(* PLC project Unnamed, Unknown Unnamed 1 *)
(* stored: creationDateTime 2025-11-24T11:16:17, modificationDateTime 2025-11-28T12:57:50 *)

PROGRAM Lab2
  VAR
    Potentiometer AT %IW1 : UINT := 1;
    Ljussensor AT %IW2 : UINT := 1;
  END_VAR
  VAR
    S0 : BOOL := False;
    S1 : BOOL := False;
    Light_sample : BOOL := False;
    Poten_sample : BOOL;
    Light_damaged : BOOL := False;
    Poten_damaged : BOOL := False;
    Dark : BOOL := False;
    Bright : BOOL := False;
    High : BOOL := False;
    Medium : BOOL := False;
    Low : BOOL := False;
    Damaged_comp : UINT := 0;
    Light_comp : UINT := 32768;
    High_comp : UINT := 43690;
    Low_comp : UINT := 21845;
  END_VAR
  VAR
    Relay AT %QX0.0 : BOOL := 0;
  END_VAR
  VAR
    CTU0 : CTU;
    TON0 : TON;
    T50ms : TIME := T#50ms;
    Tick_100ms : BOOL := 0;
    Fifty_ticks : INT := 50;
    TON1 : TON;
    R_TRIG0 : R_TRIG;
    F_TRIG0 : F_TRIG;
  END_VAR
  VAR  (* added by the conversion: wires and edge detectors of the diagram *)
    R_TRIG1 : R_TRIG;
    _GT34_OUT : BOOL;
    _LT35_OUT : BOOL;
    _EQ80_OUT : BOOL;
  END_VAR

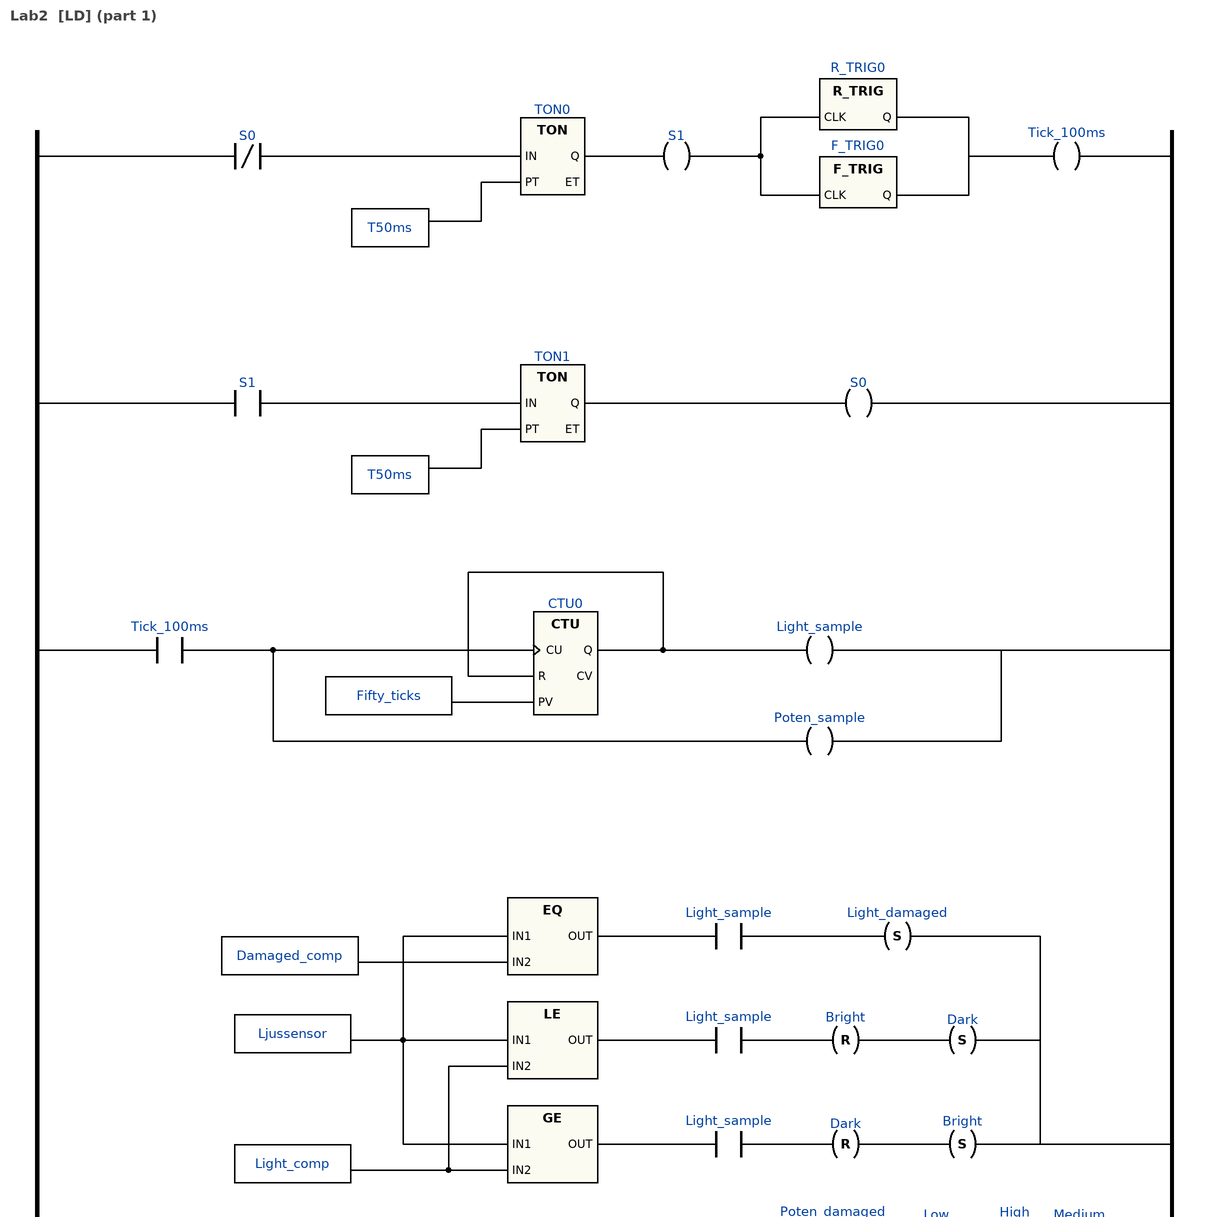
(* LD diagram, written out as Structured Text *)
TON0(IN := NOT S0, PT := T50ms);
R_TRIG0(CLK := TON0.Q);
F_TRIG0(CLK := TON0.Q);
Tick_100ms := R_TRIG0.Q OR F_TRIG0.Q;
R_TRIG1(CLK := Tick_100ms);
CTU0(CU := R_TRIG1.Q, R := CTU0.Q, PV := Fifty_ticks);
Light_sample := CTU0.Q;
TON1(IN := S1, PT := T50ms);
S0 := TON1.Q;
S1 := TON0.Q;
Poten_sample := Tick_100ms;
IF Ljussensor = Damaged_comp AND Light_sample THEN Light_damaged := TRUE; END_IF;
IF Ljussensor >= Light_comp AND Light_sample THEN Bright := TRUE; END_IF;
IF Ljussensor <= Light_comp AND Light_sample THEN Dark := TRUE; END_IF;
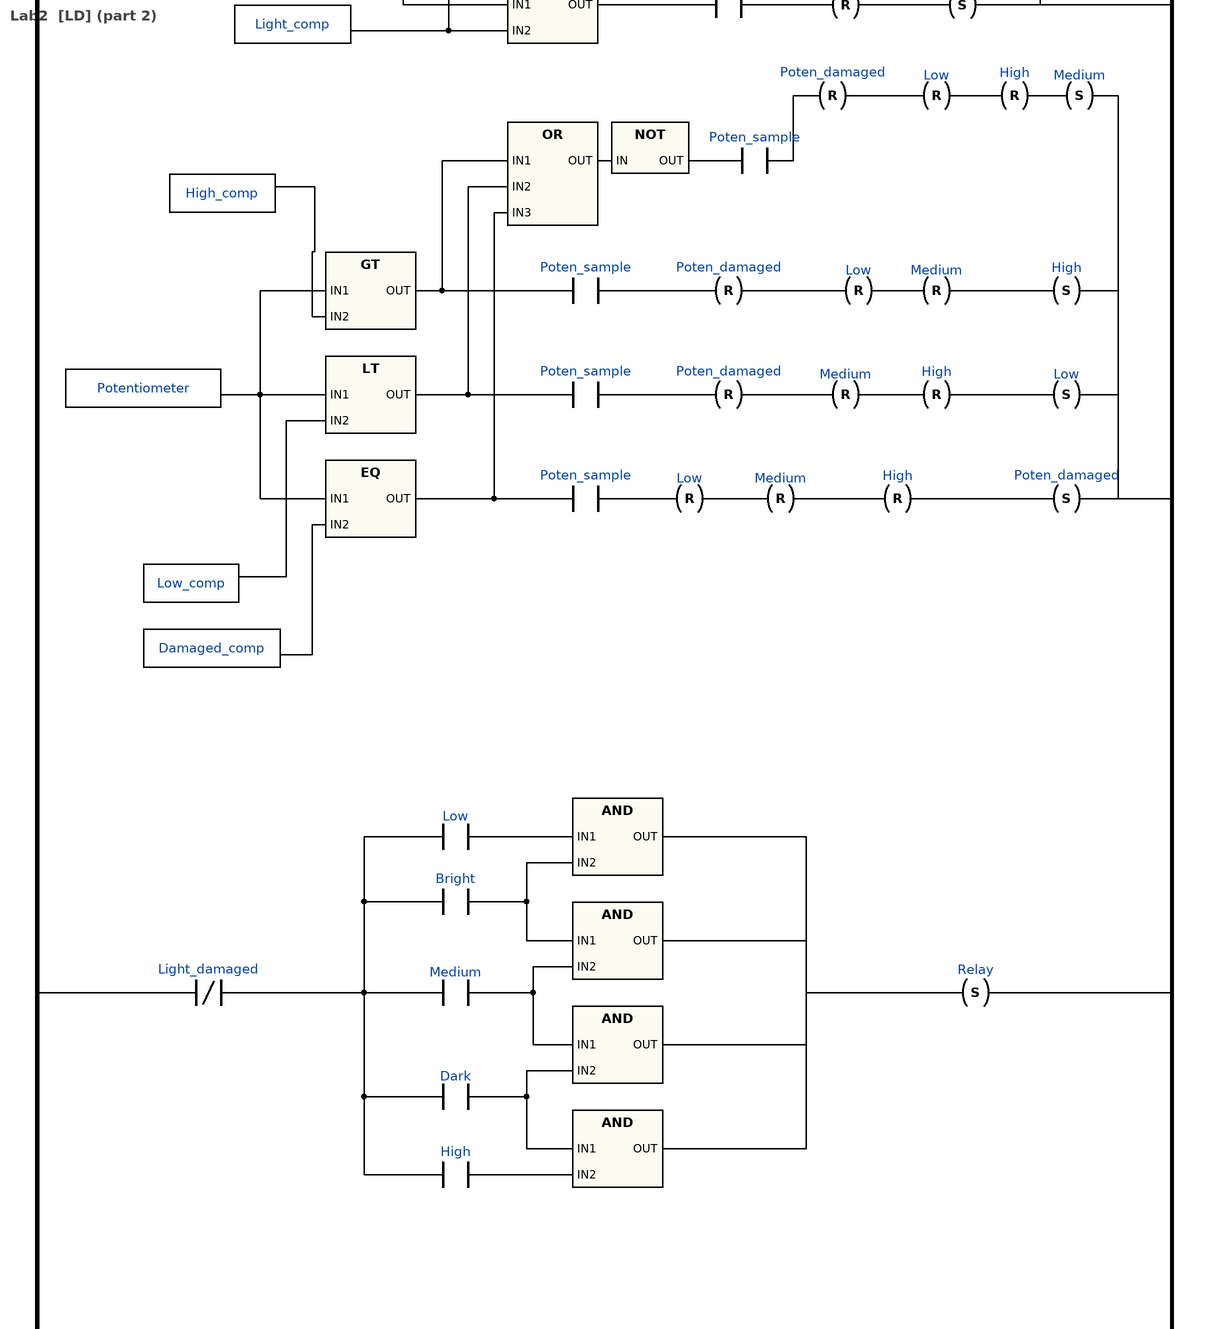
_GT34_OUT := Potentiometer > High_comp;
IF _GT34_OUT AND Poten_sample THEN High := TRUE; END_IF;
_LT35_OUT := Potentiometer < Low_comp;
IF _LT35_OUT AND Poten_sample THEN Low := TRUE; END_IF;
_EQ80_OUT := Potentiometer = Damaged_comp;
IF NOT (_GT34_OUT OR _LT35_OUT OR _EQ80_OUT) AND Poten_sample THEN Medium := TRUE; END_IF;
IF _EQ80_OUT AND Poten_sample THEN Poten_damaged := TRUE; END_IF;
IF NOT Light_damaged AND Low AND NOT Light_damaged AND Bright OR NOT Light_damaged AND Bright AND NOT Light_damaged AND Medium OR NOT Light_damaged AND Dark AND NOT Light_damaged AND High OR NOT Light_damaged AND Medium AND NOT Light_damaged AND Dark THEN Relay := TRUE; END_IF;
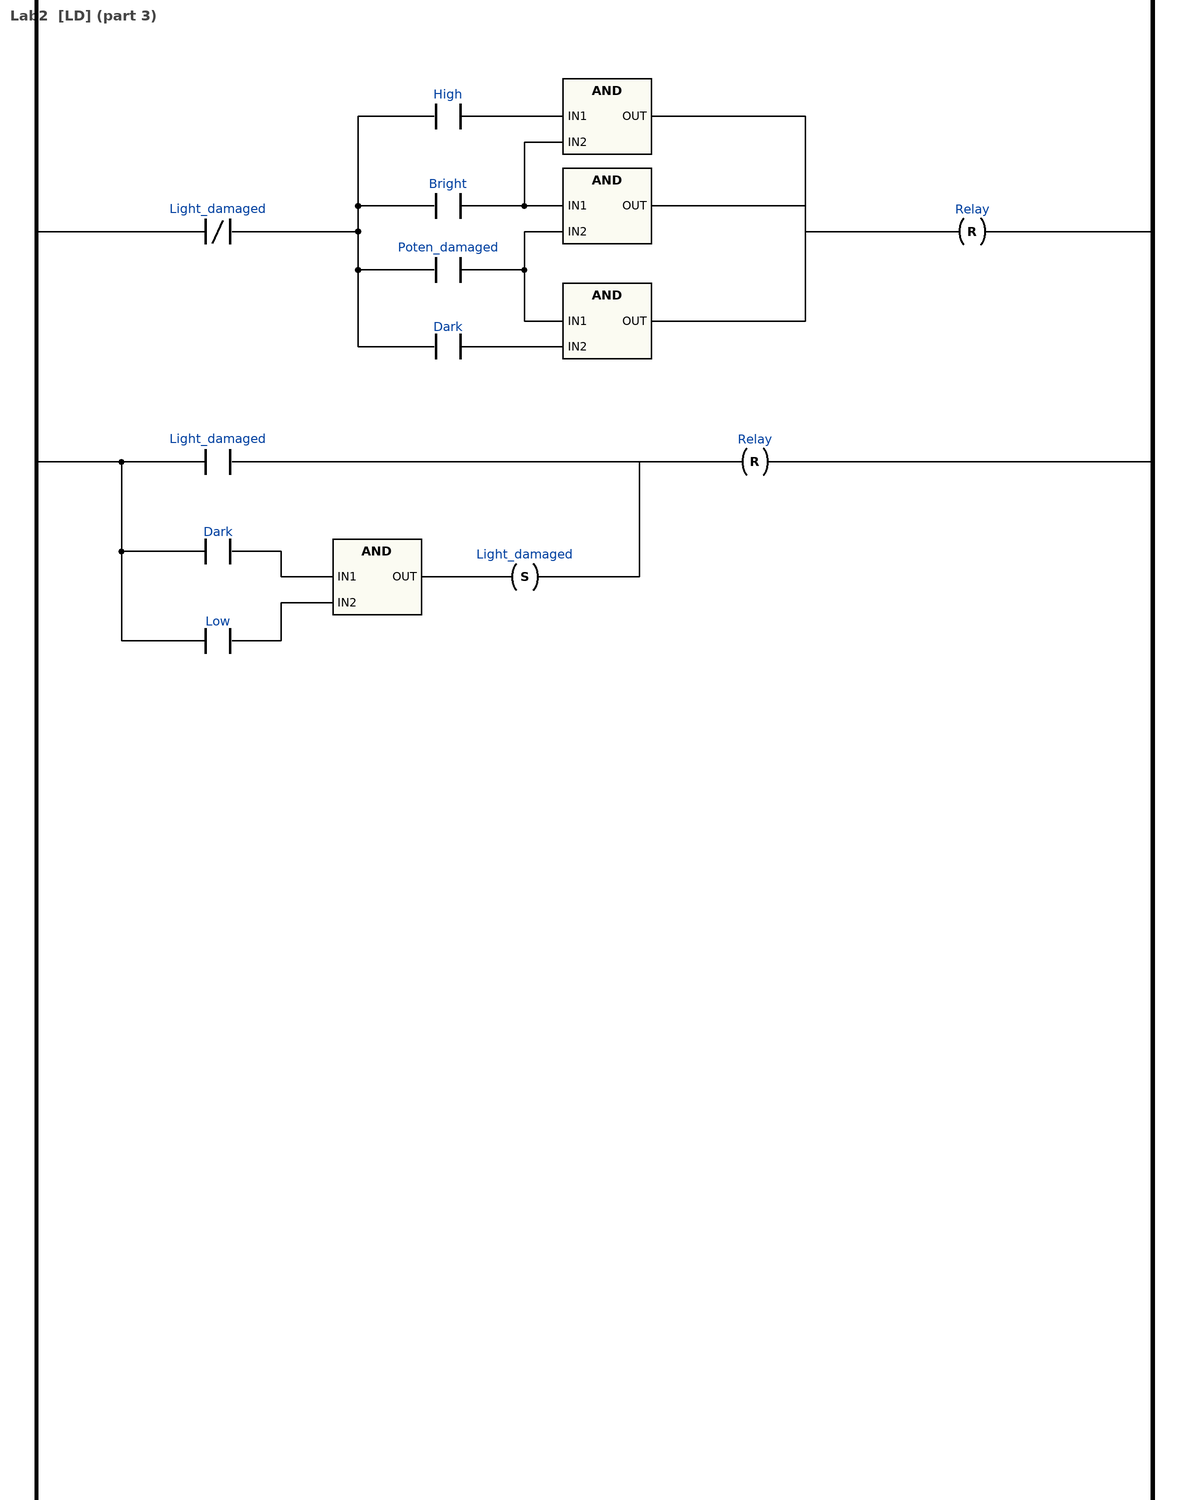
IF NOT Light_damaged AND Bright AND NOT Light_damaged AND Poten_damaged OR NOT Light_damaged AND High AND NOT Light_damaged AND Bright OR NOT Light_damaged AND Poten_damaged AND NOT Light_damaged AND Dark THEN Relay := FALSE; END_IF;
IF Light_damaged OR Dark AND Low THEN Relay := FALSE; END_IF;
IF Dark AND Low THEN Light_damaged := TRUE; END_IF;
IF Ljussensor >= Light_comp AND Light_sample THEN Dark := FALSE; END_IF;
IF Ljussensor <= Light_comp AND Light_sample THEN Bright := FALSE; END_IF;
IF _GT34_OUT AND Poten_sample THEN Poten_damaged := FALSE; END_IF;
IF _LT35_OUT AND Poten_sample THEN Poten_damaged := FALSE; END_IF;
IF NOT (_GT34_OUT OR _LT35_OUT OR _EQ80_OUT) AND Poten_sample THEN Poten_damaged := FALSE; END_IF;
IF _EQ80_OUT AND Poten_sample THEN Low := FALSE; END_IF;
IF _GT34_OUT AND Poten_sample THEN Low := FALSE; END_IF;
IF NOT (_GT34_OUT OR _LT35_OUT OR _EQ80_OUT) AND Poten_sample THEN Low := FALSE; END_IF;
IF _GT34_OUT AND Poten_sample THEN Medium := FALSE; END_IF;
IF _LT35_OUT AND Poten_sample THEN Medium := FALSE; END_IF;
IF _EQ80_OUT AND Poten_sample THEN Medium := FALSE; END_IF;
IF NOT (_GT34_OUT OR _LT35_OUT OR _EQ80_OUT) AND Poten_sample THEN High := FALSE; END_IF;
IF _LT35_OUT AND Poten_sample THEN High := FALSE; END_IF;
IF _EQ80_OUT AND Poten_sample THEN High := FALSE; END_IF;
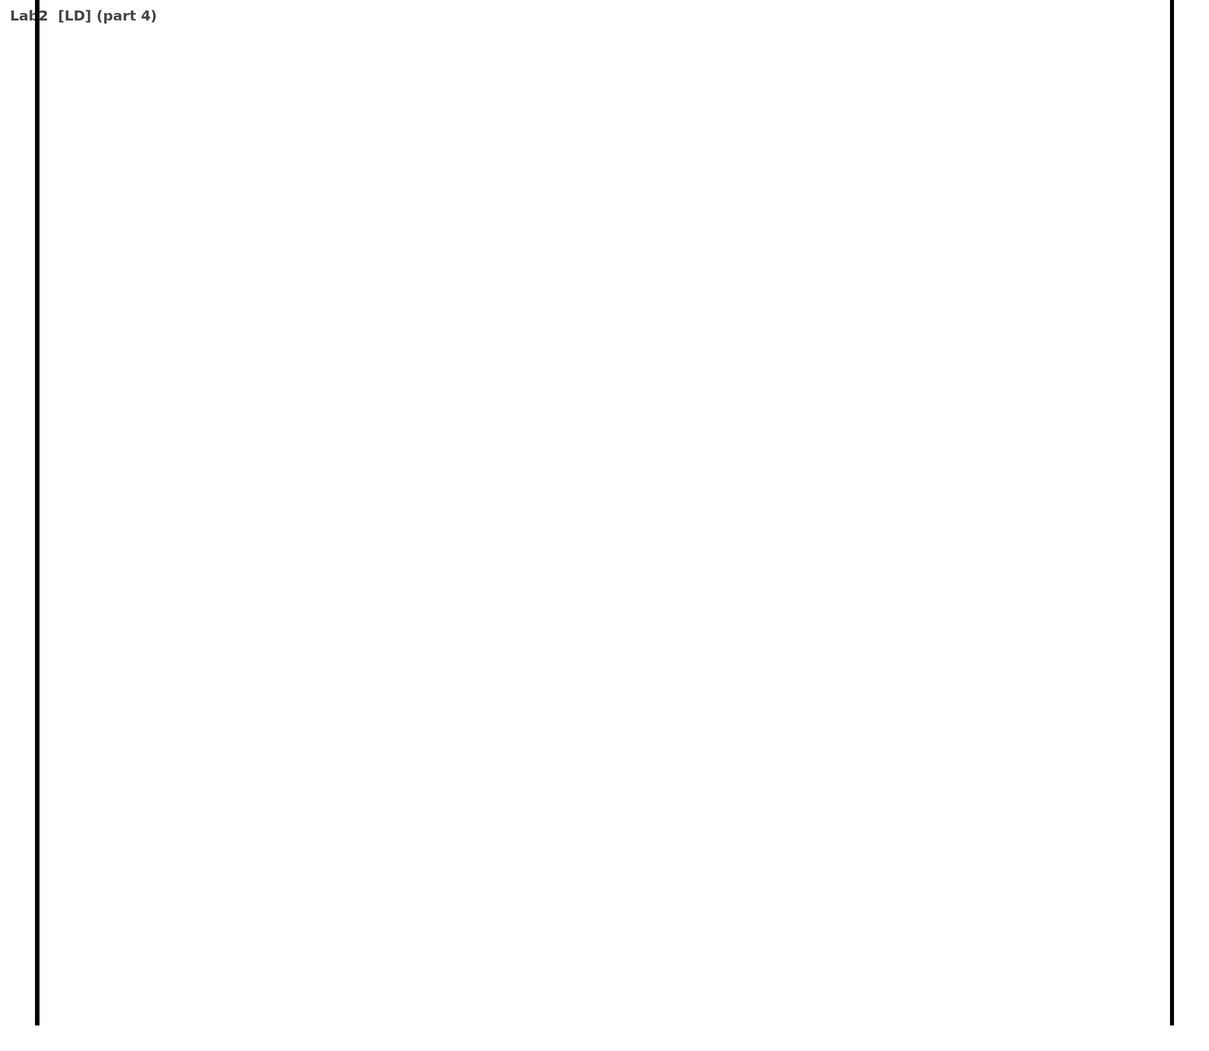
END_PROGRAM

CONFIGURATION Config0
  RESOURCE Res0 ON PLC
    TASK task0(INTERVAL := T#20ms, PRIORITY := 0);
    PROGRAM instance0 WITH task0 : Lab2;
  END_RESOURCE
END_CONFIGURATION
